FUNCTION_BLOCK LOADFORECASTER_DEB (* Function block for holding historical PV power measurements and generating PV power forecasts. *)
  (* Standard: 61499-2; Description: IEC 61499 implementation of the "PVprog" algorithm. Original version's MIT license: Copyright (c) 2016 Joseph Bergner, Johannes Weniger, Tjarko Tjaden Permission is hereby granted, free of charge, to any person obtaining a copy of this software and associated documentation files (the "Software"), to deal in the Software without restriction, including without limitation the rights to use, copy, modify, merge, publish, distribute, sublicense, and/or sell copies of the Software, and to permit persons to whom the Software is furnished to do so, subject to the following conditions: The above copyright notice and this permission notice shall be included in all copies or substantial portions of the Software. THE SOFTWARE IS PROVIDED "AS IS", WITHOUT WARRANTY OF ANY KIND, EXPRESS OR IMPLIED, INCLUDING BUT NOT LIMITED TO THE WARRANTIES OF MERCHANTABILITY, FITNESS FOR A PARTICULAR PURPOSE AND NONINFRINGEMENT. IN NO EVENT SHALL THE AUTHORS OR COPYRIGHT HOLDERS BE LIABLE FOR ANY CLAIM, DAMAGES OR OTHER LIABILITY, WHETHER IN AN ACTION OF CONTRACT, TORT OR OTHERWISE, ARISING FROM, OUT OF OR IN CONNECTION WITH THE SOFTWARE OR THE USE OR OTHER DEALINGS IN THE SOFTWARE. *)
  (* Version 0.0, 2017-05-03, 4DIAC-IDE, 4DIAC-Consortium *)
  (* Version 1.0, 2017-05-03, Marc Jakobi, HTW Berlin *)
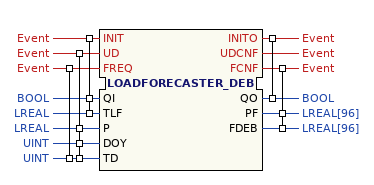
  EVENT_INPUT
    INIT WITH QI, TLF; (* Initialization Request *)
    UD WITH P, TD, DOY; (* PV Forecast Update Request *)
    FREQ WITH TD; (* Forecast Request *)
  END_EVENT
  EVENT_OUTPUT
    INITO WITH QO; (* Initialization Confirm *)
    UDCNF; (* Update Algorithm Execution Confirmation *)
    FCNF WITH PF, FDEB; (* Forecast Confirmation *)
  END_EVENT
  VAR_INPUT
    QI : BOOL; (* Input event qualifier *)
    TLF : LREAL := 15; (* Time frame to forecast ahead (and look back) in h *)
    P : LREAL; (* Measured PV power in W *)
    DOY : UINT := 1; (* Day of the year [1..365] *)
    TD : UINT := 0; (* Time of day [min] [0..1439] *)
  END_VAR
  VAR_OUTPUT
    QO : BOOL; (* Output event qualifier *)
    PF : ARRAY [0..95] OF LREAL; (* Forecasted Load *)
    FDEB : ARRAY [0..95] OF LREAL; (* Forecast debug output *)
  END_VAR
  VAR
    LOOKBACKTIMEINTIMESTEPS : UINT; (* Number of time steps (minutes) to look back when generating forecasts *)
    LOOKFORWARDTIMEINTIMESTEPS : UINT; (* Number of time steps (15 min intervals) to look ahead for forecast *)
    LOOKBACKTIMEINHOURS : LREAL; (* Time frame to look back when generating forecasts in h *)
    LOOKFORWARDTIMEINHOURS : LREAL; (* Time frame to forecast ahead in h *)
    POWERLASTDAY : ARRAY [0..1439] OF LREAL; (* Stores the historical PV power [W] of the last day *)
    POWERCURRDAY : ARRAY [0..1439] OF LREAL; (* Stores the historical PV power [W] of the current day *)
    LASTTIMESTEP : INT := -1; (* Time at the point of the last call of the prepareForecast algorithm *)
    LASTDAYOFYEAR : UINT := 0; (* Day of the year [1...365] of the last call of the prepareForecast algorithm *)
    TIMESINCELASTUPDATE : INT := 1; (* Time [min] between last update and current one *)
    LASTMEASUREDPOWER : LREAL := 0; (* Power P [W] input when last update occurred *)
    PU : LREAL := 0; (* Power (either current or interpolated) [W] used for updating memory *)
    TIMEINDEX : UINT := 0; (* Time index (either current or interpolated) [min] used for updating memory *)
    LONGTERMWEIGHT : ARRAY [0..1439] OF LREAL; (* Function for the variable weighting of the long term persistence forecast over the forecast horizon [0,...1] *)
    SHORTTERMWEIGHT : ARRAY [0..1439] OF LREAL; (* Function for the variable weighting of the short term persistence forecast over the forecast horizon [0,...1] *)
    LOAD15MEANCURRDAY : ARRAY [0..95] OF LREAL; (* 15 minute running mean of the load [W] of the current day *)
    LOAD15MEANLASTDAY : ARRAY [0..95] OF LREAL; (* 15 minute running mean of the load [W] of the day preceeding the current day *)
    TLB : LREAL := 15; (* Time frame to look back when generating forecasts in h *)
  END_VAR
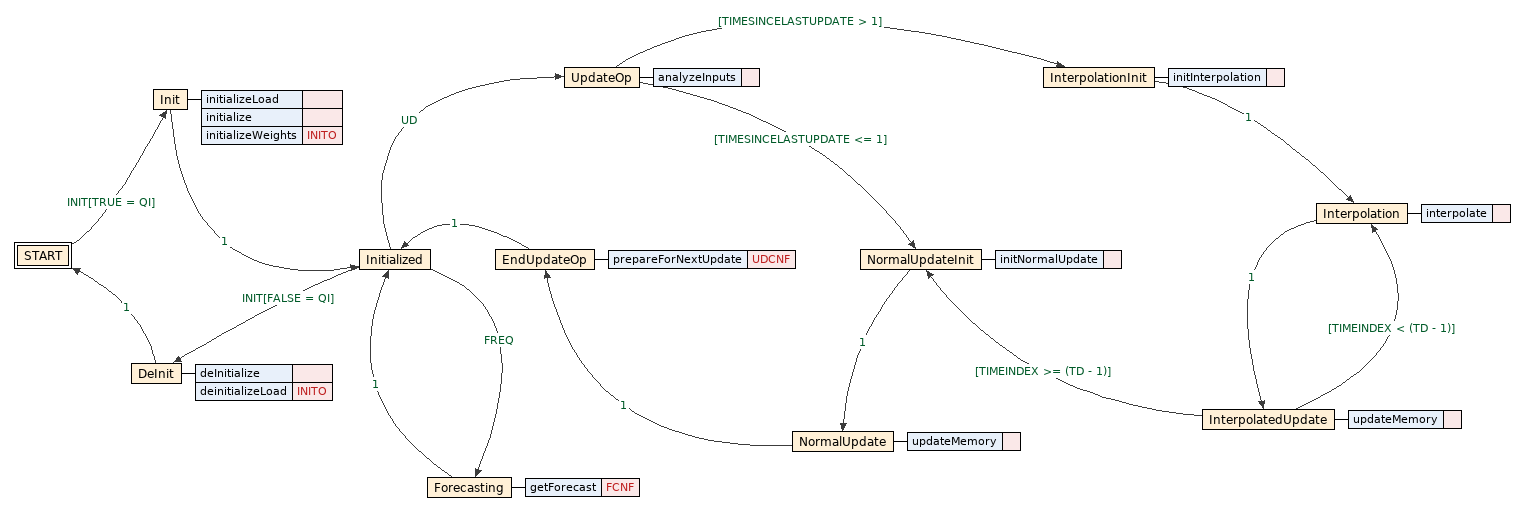
  EC_STATES
    START; (* Initial State *)
    Init : initializeLoad, initialize, initializeWeights -> INITO; (* Initialization *)
    UpdateOp : analyzeInputs; (* Normal execution *)
    Initialized;
    DeInit : deInitialize, deinitializeLoad -> INITO;
    Forecasting : getForecast -> FCNF;
    Interpolation : interpolate;
    NormalUpdate : updateMemory;
    EndUpdateOp : prepareForNextUpdate -> UDCNF;
    InterpolatedUpdate : updateMemory;
    NormalUpdateInit : initNormalUpdate;
    InterpolationInit : initInterpolation;
  END_STATES
  EC_TRANSITIONS
    DeInit TO START := 1;
    START TO Init := INIT[TRUE = QI];
    Init TO Initialized := 1;
    Initialized TO DeInit := INIT[FALSE = QI];
    Forecasting TO Initialized := 1;
    Initialized TO Forecasting := FREQ;
    Initialized TO UpdateOp := UD;
    EndUpdateOp TO Initialized := 1;
    NormalUpdate TO EndUpdateOp := 1;
    UpdateOp TO NormalUpdateInit := [TIMESINCELASTUPDATE <= 1];
    UpdateOp TO InterpolationInit := [TIMESINCELASTUPDATE > 1];
    InterpolationInit TO Interpolation := 1;
    Interpolation TO InterpolatedUpdate := 1;
    InterpolatedUpdate TO Interpolation := [TIMEINDEX < (TD - 1)];
    InterpolatedUpdate TO NormalUpdateInit := [TIMEINDEX >= (TD - 1)];
    NormalUpdateInit TO NormalUpdate := 1;
  END_TRANSITIONS
  ALGORITHM initialize IN ST: (* Initialization algorithm *)
VAR
	tmp1 : LREAL;
	tmp2 : UINT;
END_VAR;
/*
 * Used internal vars & inputs:
 * TLB, TLF, LOOKBACKTIMEINHOURS, LOOKFORWARDTIMEINHOURS : LREAL;
 * LOOKBACKTIMEINTIMESTEPS, LOOKFORWARDTIMEINTIMESTEPS : UINT;
 * QO : BOOL;
 */
// Limit inputs to acceptable boundaries
IF TLB < 0 THEN
	TLB := 0;
ELSIF TLB > 24 THEN
	TLB := 24;
END_IF;
LOOKBACKTIMEINHOURS := TLB;
// Workaround for ceil function
tmp1 := LOOKBACKTIMEINHOURS * 60; // input resolution = 1 min
tmp2 := LREAL_TO_UINT(tmp1);
IF UINT_TO_LREAL(tmp2) < tmp1 THEN
 	LOOKBACKTIMEINTIMESTEPS := tmp2 + 1;
ELSE
	LOOKBACKTIMEINTIMESTEPS := tmp2;
END_IF;
// Set forecast horizon
IF TLF < 0 THEN
	TLF := 0;
ELSIF TLF > 24 THEN
	TLF := 24;
END_IF;
LOOKFORWARDTIMEINHOURS := TLF;
tmp1 := LOOKFORWARDTIMEINHOURS * 4; // output resolution = 15 min
tmp2 := LREAL_TO_UINT(tmp1);
IF UINT_TO_LREAL(tmp2) < tmp1 THEN
 	LOOKFORWARDTIMEINTIMESTEPS := tmp2 + 1;
ELSE
	LOOKFORWARDTIMEINTIMESTEPS := tmp2;
END_IF;
QO := QI; // Pass Input event qualifier to output event qualifier
  END_ALGORITHM
  ALGORITHM deInitialize IN ST: (* Deinitialization algorithm *)
VAR
	j : UINT;
END_VAR;
/*
 * Used internal vars & inputs:
 * POWERCURRDAY, POWERLASTDAY, LASTMEASUREDPOWER : LREAL;
 * LASTDAYOFYEAR : UINT;
 * LASTTIMESTEP : INT;
 * QO : BOOL;
 */
// Reset all internal variables to initial values
FOR j := 0 TO 1439 BY 1 DO
	POWERCURRDAY[j] := 0;
	POWERLASTDAY[j] := 0;
END_FOR;
LASTDAYOFYEAR := 0;
LASTTIMESTEP := -1;
LASTMEASUREDPOWER := 0;
QO := FALSE;
  END_ALGORITHM
  ALGORITHM analyzeInputs IN ST: (* Stores load data and prepares it for forecast generation *)
VAR
	i : UINT;
END_VAR;
/*
 * Used internal vars & inputs:
 * DOY, LASTDAYPFYEAR, TD : UINT;
 * TIMESINCELASTUPDATE, LASTTIMESTEP : INT;
 * POWERLASTDAY, POWERCURRDAY, LOAD15MEANLASTDAY, LOAD15MEANCURRDAY : LREAL;
 */
TIMESINCELASTUPDATE := UINT_TO_INT(TD) - LASTTIMESTEP;
// At the beginning of each day, replace LASTDAY arrays with CURRDAY arrays
IF DOY <> LASTDAYOFYEAR THEN
	FOR i := 0 TO 1439 BY 1 DO
		POWERLASTDAY[i] := POWERCURRDAY[i];
	END_FOR;
	FOR i := 0 TO 95 BY 1 DO
		LOAD15MEANLASTDAY[i] := LOAD15MEANCURRDAY[i];
	END_FOR;
	LASTDAYOFYEAR := DOY;
	TIMESINCELASTUPDATE := 1; // Set to 1 minute for beginning of day
END_IF;
  END_ALGORITHM
  ALGORITHM getForecast IN ST: (* Generates forecast from currently stored load data *)
VAR
	forecastIndex : UINT;
	td15 : UINT;
	j : INT;
	tmpI : INT;
	shortTermPower : LREAL;
	longTermPower : LREAL;
END_VAR;
/*
 * Used internal vars & inputs:
 * DOY, TD, LOOKFORWARDTIMEINTIMESTEPS : UINT;
 * PF, LOAD15MEANCURRDAY, LOAD15MEANLASTDAY, SHORTTERMWEIGHT, LONGTERMWEIGHT : LREAL;
 */
td15 := TD / 15; // Time of day in 15 min intervals
// Calculate 15 minute mean of POWERCURRDAY
LOAD15MEANCURRDAY[td15]  := POWERCURRDAY[TD];
// tmpI := MAX(0, TD - 16);
tmpI := UINT_TO_INT(TD) -  16; // Temporary variable for setting loop index's lower limit to 0
IF tmpI < 0 THEN
	tmpI := 0;
END_IF;
FOR j := tmpI TO UINT_TO_INT(TD) - 1 BY 1 DO
	LOAD15MEANCURRDAY[td15]  := LOAD15MEANCURRDAY[td15]  + POWERCURRDAY[j];
END_FOR;
LOAD15MEANCURRDAY[td15]  := LOAD15MEANCURRDAY[td15]  / 15;
// Multiply weighting functions with the persistence forecasts to generate load forecast
IF TD > 0 THEN
	shortTermPower := LOAD15MEANCURRDAY[td15 - 1];
ELSE
	shortTermPower := LOAD15MEANLASTDAY[95]; // Last cached value of yesterday
END_IF;
forecastIndex := 0;
// Look back 96 steps
// 96 * (15 + 1 - 15) = 96 * 1 = 96
FOR j := UINT_TO_INT(td15) - 96 TO UINT_TO_INT(td15) - (96 - UINT_TO_INT(LOOKFORWARDTIMEINTIMESTEPS)) - 1 BY 1 DO
	IF j < 0 THEN
		longTermPower := LOAD15MEANLASTDAY[ j + 96];
	ELSE
		longTermPower := LOAD15MEANCURRDAY[j];
	END_IF;
	PF[forecastIndex] := LONGTERMWEIGHT[forecastIndex] * longTermPower + SHORTTERMWEIGHT[forecastIndex] * shortTermPower;
	forecastIndex := forecastIndex + 1;
END_FOR;
  END_ALGORITHM
  ALGORITHM updateMemory IN ST: (* Updates the memory with measured or interpolated PV data *)
/*
 * Used internal vars & inputs:
 * POWERCURRDAY, PU  : LREAL;
 * TIMEINDEX  : UINT;
 */
POWERCURRDAY[TIMEINDEX] := PU;
  END_ALGORITHM
  ALGORITHM interpolate IN ST: (* Interpolates between last and currently measured PV data *)
/*
 * Used internal vars & inputs:
 * INTERPOLATIONINCREMENT, LASTMEASUREDPOWER, P, PU  : LREAL;
 * TD, TIMEINDEX  : UINT;
 */
// Linear interpolation between last measured power and currently measured power
PU := PU + (P - LASTMEASUREDPOWER) / INT_TO_LREAL(TIMESINCELASTUPDATE);
TIMEINDEX := TIMEINDEX + 1;
  END_ALGORITHM
  ALGORITHM prepareForNextUpdate IN ST: (* Saves the current inputs for next update *)
/*
 * Used internal vars & inputs:
 * LASTMEASUREDPOWER : LREAL;
 * LASTTIMESTEP : INT;
 * TD : UINT;
 */
LASTMEASUREDPOWER := P;
LASTTIMESTEP := UINT_TO_INT(TD);
  END_ALGORITHM
  ALGORITHM initNormalUpdate IN ST: (* Sets memory update inputs PU and TIMEINDEX to current values *)
/*
 * Used internal vars & inputs:
 * P, PU : LREAL;
 * TD, TIMEINDEX : UINT;
 */
PU := P;
TIMEINDEX := TD;
  END_ALGORITHM
  ALGORITHM initInterpolation IN ST: (* Sets tieme index to initialize interpolation *)
/*
 * Used internal vars & inputs:
 * TD, TIMEINDEX : UINT;
 * TIMESINCELASTUPDATE : INT;
 * LASTMEASUREDPOWER, PU : LREAL;
 */
 // Initialize TIMEINDEX and PU for interpolation
TIMEINDEX := TD - INT_TO_UINT(TIMESINCELASTUPDATE) + 1;
PU := LASTMEASUREDPOWER;
  END_ALGORITHM
  ALGORITHM initializeWeights IN ST: (* Algorithm for initializing the weighting functions LONGTERMWEIGHT and SHORTTERMWEIGHT *)
VAR
	i : UINT;
	tmp1 : LREAL;
	tmp2 : LREAL;
END_VAR;
/*
 * Used internal vars & inputs:
 * SHORTTERMWEIGHT, LONGTERMWEIGHT, EULER : LREAL;
 * LOOKFORWARDTIMEINTIMESTEPS : UINT;
 */
tmp1 := 0.1; // must be defined here to prevent EXP function ambiguity
FOR i := 0 TO LOOKFORWARDTIMEINTIMESTEPS - 1 BY 1 DO
	tmp2 := -0.1 * (UINT_TO_LREAL(i) + 1); // must be defined here to prevent EXP function ambiguity
	SHORTTERMWEIGHT[i] := 1 / EXP(tmp1) * EXP(tmp2);
	LONGTERMWEIGHT[i] := 1 - SHORTTERMWEIGHT[i];
END_FOR;
  END_ALGORITHM
  ALGORITHM deinitializeLoad IN ST: (* LoadForecaster-specific deinitilization algorithm *)
VAR
	i : UINT;
END_VAR;
/*
 * Used internal vars & inputs:
 * LOAD15MEANCURRDAY, LOAD15MEANLASTDAY : LREAL;
 */
 FOR i := 0 TO 95 BY 1 DO
 	LOAD15MEANCURRDAY[i] := 0;
 	LOAD15MEANLASTDAY[i] := 0;
 END_FOR;
  END_ALGORITHM
  ALGORITHM initializeLoad IN ST: (* LoadForecaster-specific initialization algorithm: Sets lookback time equal to look-forward time. *)
/*
 * Used internal vars & inputs:
 * TLB, TLF : LREAL;
 */
TLB := TLF;
  END_ALGORITHM
END_FUNCTION_BLOCK
